FUNCTION_BLOCK FINAL FindJsonMember IMPLEMENTS Callback
VAR_INPUT
	memberToFind: STRING;
	jsonDomParser: REFERENCE TO FB_JsonDomParser;
	jsonReference: REFERENCE TO SJsonValue;
	memberReference: REFERENCE TO SJsonValue;
END_VAR


(* This is method get's exectued by the framework when the callback is triggered.
 It returns a step number which might be used together with Await to jump to a certain chain step
 after the callback code has been executed.*)
METHOD execute : UDINT
memberReference := jsonDomParser.FindMember(jsonReference, memberToFind);
END_METHOD

END_FUNCTION_BLOCK

(* stored: Version 1.1.0.1, ProductVersion 3.1.4024.12
   POU FindJsonMember: Id {f31b7faf-314c-45d4-9960-c055c68f91e9}, SpecialFunc None
   Method execute: Id {251b2f64-dc0e-43ca-b866-3276e4e297a6} *)
